TYPE sc_db_Steel_Status :
STRUCT
	uuid : STRING(36);
	steel_status : STRING(80);
	steel_location : STRING(80);
END_STRUCT
END_TYPE

(* stored: Version 1.1.0.1, ProductVersion 3.1.4026.13
   DUT sc_db_Steel_Status: Id {ebfeb098-7626-4d0c-b90b-32be502bed7e} *)
